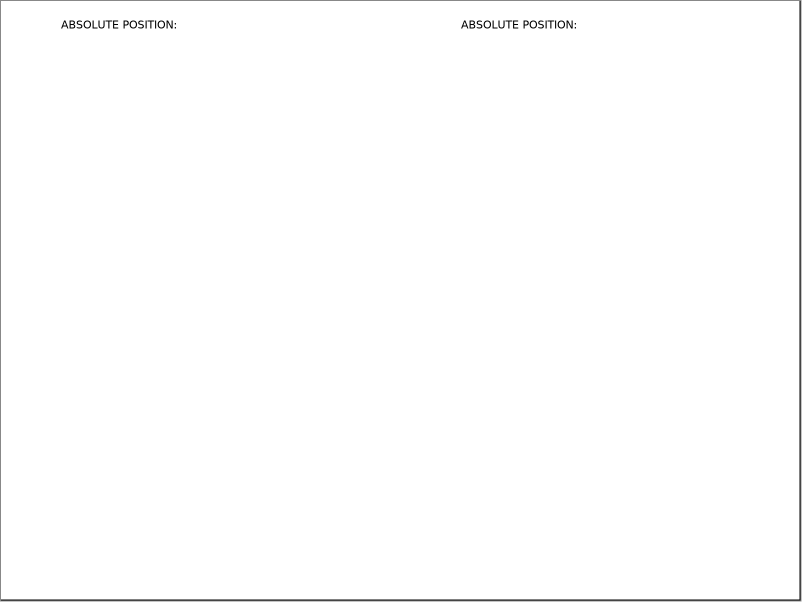
VISUALIZATION F18_Set_Override  // 802x602
    Rectangle (0,0 800x600)
    Label (10,10 170x30), "ABSOLUTE POSITION:"
    Label (410,10 170x30), "ABSOLUTE POSITION:"
END_VISUALIZATION

(* stored: Version 1.1.0.1, ProductVersion 3.1.4022.7
   Visu F18_Set_Override: Id {ce0e7b7b-12d0-4a68-93ba-69e425b88c99} *)
